   REGION "Manipolatori - Movimento BTrk da Uscita Deposito A0303 alto Vs Uscita deposito A0303 basso"
      "BTrk_Presence"(
         en := TRUE,
         Item := BTrk.A0302_EXIT.B
      );

      "BTrk_Absence"(
         en := "BTrk_Presence"(Item := BTrk.A0302_EXIT.B),
         Item := BTrk.A0302_EXIT.B
      );

      "BTrk_Absence"(
         en := "BTrk_Absence"(Item := BTrk.A0302_EXIT.B),
         Item := BTrk.A0303.Preparation.B
      );

      "BTrk_Presence"(
         en := BTrk.A0302_EXIT.B,
         Item := BTrk.A0302_EXIT.B
      );

      "BTrk_Presence"(Item := BTrk.A0302_EXIT.B);
      IF "BTrk_Presence"(Item := BTrk.A0302_EXIT.B) THEN
         "BTrk_Absence"(Item := BTrk.A0302_EXIT.B);
      END_IF;
      IF "BTrk_Absence"(Item := BTrk.A0302_EXIT.B) THEN
         "BTrk_Absence"(Item := BTrk.A0303.Preparation.B);
      END_IF;
      Ctrl.TRK.BTrk.CheckOut_GoodQlty_UP_To_DOWN := ((("BTrk_Absence"(Item := BTrk.A0303.Preparation.B) AND CIn.Manipolatori.InPos_BancoA0303) AND CIn.Banco_A0303.ReadyToRecive) OR (("BTrk_Absence"(Item := BTrk.A0303.Preparation.B) AND CIn.Manipolatori.InPos_BancoA0303) AND A03_DEBUG.A0302_Manager.A0303_ReadyToRecive));
      IF ((Ctrl.TRK.BTrk.CheckOut_GoodQlty_UP_To_DOWN AND CIn.Manipolatori.Testa.Sollevatore.Work) AND CIn.Manipolatori.Coda.Sollevatore.Work) THEN
         BTrk.A0302_EXIT.B := BTrk.A0302_EXIT.B;
      END_IF;
   END_REGION

   REGION "Manipolatori - Movimento BTrk  Uscita deposito A0303 basso == a ==> Rilascia Beam"
      "BTrk_Presence"(
         en := TRUE,
         Item := BTrk.A0302_EXIT.B
      );

      "BTrk_Absence"(
         en := "BTrk_Presence"(Item := BTrk.A0302_EXIT.B),
         Item := BTrk.A0303.Preparation.B
      );

      "BTrk_Presence"(Item := BTrk.A0302_EXIT.B);
      IF "BTrk_Presence"(Item := BTrk.A0302_EXIT.B) THEN
         "BTrk_Absence"(Item := BTrk.A0303.Preparation.B);
      END_IF;
      Ctrl.TRK.BTrk.CheckOut_GoodQlty_DOWN_To_Sgancia := (((("BTrk_Absence"(Item := BTrk.A0303.Preparation.B) AND CIn.Manipolatori.Testa.Sollevatore.Rest) AND CIn.Manipolatori.Coda.Sollevatore.Rest) AND CIn.Manipolatori.Testa.Sollevatore.Standstill) AND CIn.Manipolatori.Coda.Sollevatore.Standstill);
      IF ((((Ctrl.TRK.BTrk.CheckOut_GoodQlty_DOWN_To_Sgancia AND CIn.Manipolatori.Testa.Magnete.Rest) AND CIn.Manipolatori.Coda.Magnete.Rest) AND NOT (CIn.CarroPareggTesta.Sens.PresenzaMat)) AND NOT (CIn.CarroPareggCoda.Sens.PresenzaMat)) THEN
         BTrk.A0303.Preparation.B := BTrk.A0302_EXIT.B;
      END_IF;
   END_REGION

   REGION "[Ax] Manipolatore - Control - Pos. PRELIEVO su carri pareggiatori"
      "BTrk_Absence"(
         en := TRUE,
         Item := BTrk.A0302_EXIT.B
      );

      "BTrk_Absence"(
         en := "BTrk_Absence"(Item := BTrk.A0302_EXIT.B),
         Item := BTrk.A0302_EXIT.B
      );

      "BTrk_Absence"(
         en := "BTrk_Absence"(Item := BTrk.A0302_EXIT.B),
         Item := BTrk.A0302_EXIT.B
      );

      "BTrk_Absence"(
         en := "BTrk_Absence"(Item := BTrk.A0302_EXIT.B),
         Item := BTrk.A0302_EXIT.B
      );

      "BTrk_Absence"(Item := BTrk.A0302_EXIT.B);
      Ctrl.TRK.BTrk.Manipolatori_Return_ToPrelievo := ((("BTrk_Absence"(Item := BTrk.A0302_EXIT.B) AND NOT (CIn.Manipolatori.InPos_Prelievo)) AND NOT (CIn.CarroPareggCoda.Sens.PresenzaMat)) AND NOT (CIn.CarroPareggTesta.Sens.PresenzaMat));
   END_REGION

   REGION "Manipolatori - Controllo del pezzo sui Magneti - Allarme grave se perdo i sensori presenza"
      "BTrk_Presence"(
         en := TRUE,
         Item := BTrk.A0302_EXIT.B
      );

      "BTrk_Presence"(
         en := TRUE,
         Item := BTrk.A0302_EXIT.B
      );

      "BTrk_Presence"(
         en := TRUE,
         Item := BTrk.A0302_EXIT.B
      );

      #TON_AlarmWrongReadPz_Manip(
         IN := (((((((("BTrk_Presence"(Item := BTrk.A0302_EXIT.B) OR "BTrk_Presence"(Item := BTrk.A0302_EXIT.B) OR "BTrk_Presence"(Item := BTrk.A0302_EXIT.B)) AND CIn.Manipolatori.Testa.Sollevatore.Rest) AND CIn.Manipolatori.Coda.Sollevatore.Rest) AND CIn.Manipolatori.Testa.Magnete.Work) AND CIn.Manipolatori.Coda.Magnete.Work) AND NOT (CIn.CarroPareggCoda.Sens.PresenzaMat)) AND CIn.CarroPareggTesta.Sens.PresenzaMat) OR ((((((("BTrk_Presence"(Item := BTrk.A0302_EXIT.B) OR "BTrk_Presence"(Item := BTrk.A0302_EXIT.B) OR "BTrk_Presence"(Item := BTrk.A0302_EXIT.B)) AND CIn.Manipolatori.Testa.Sollevatore.Rest) AND CIn.Manipolatori.Coda.Sollevatore.Rest) AND CIn.Manipolatori.Testa.Magnete.Work) AND CIn.Manipolatori.Coda.Magnete.Work) AND CIn.CarroPareggCoda.Sens.PresenzaMat) AND NOT (CIn.CarroPareggTesta.Sens.PresenzaMat))),
         PT := T#2S
      );

      "BTrk_Presence"(Item := BTrk.A0302_EXIT.B);
      #TON_AlarmWrongReadPz_Manip.Q;
      IF #TON_AlarmWrongReadPz_Manip.Q THEN
         Alarm.WrongReadPz_ManipBasso := TRUE;
      END_IF;
   END_REGION

   REGION "[Sollevatori] - Manipolatori Testa/Coda - Movimento operazione a lavoro / a riposo"
      "BTrk_Presence"(
         en := TRUE,
         Item := BTrk.A0302_EXIT.B
      );

      "BTrk_Presence"(
         en := TRUE,
         Item := BTrk.A0302_EXIT.B
      );

      "BTrk_Presence"(
         en := TRUE,
         Item := BTrk.A0302_EXIT.B
      );

      "BTrk_Presence"(
         en := CIn.Manipolatori.InPos_BancoA0303,
         Item := BTrk.A0302_EXIT.B
      );

      "BTrk_Presence"(
         en := TRUE,
         Item := BTrk.A0302_EXIT.B
      );

      "BTrk_Presence"(Item := BTrk.A0302_EXIT.B);
      Ctrl.Manipolatori.Sollevatori.Work := ((("BTrk_Presence"(Item := BTrk.A0302_EXIT.B) OR "BTrk_Presence"(Item := BTrk.A0302_EXIT.B) OR "BTrk_Presence"(Item := BTrk.A0302_EXIT.B)) AND CIn.Manipolatori.InPos_Prelievo) OR ("BTrk_Presence"(Item := BTrk.A0302_EXIT.B) AND CIn.Banco_A0303.ReadyToRecive) OR (("BTrk_Presence"(Item := BTrk.A0302_EXIT.B) AND NOT (CIn.Manipolatori.Testa.Magnete.Rest)) AND NOT (CIn.Manipolatori.Coda.Magnete.Rest)));
      IF ((NOT (CIn.Manipolatori.InPos_BancoA0303) AND NOT (CIn.Manipolatori.InPos_Prelievo)) AND NOT (CIn.Manipolatori.InPos_BancoScarto)) THEN
         Ctrl.Manipolatori.Sollevatori.Work := FALSE;
      END_IF;
      Ctrl.Manipolatori.Sollevatori.Rest := NOT (Ctrl.Manipolatori.Sollevatori.Work);
   END_REGION

   REGION "[Magneti] - Manipolatori Testa/Coda - Movimento operazione a lavoro / a riposo"
      "BTrk_Presence"(
         en := TRUE,
         Item := BTrk.A0302_EXIT.B
      );

      "BTrk_Presence"(
         en := TRUE,
         Item := BTrk.A0302_EXIT.B
      );

      "BTrk_Presence"(
         en := TRUE,
         Item := BTrk.A0302_EXIT.B
      );

      "BTrk_Presence"(
         en := TRUE,
         Item := BTrk.A0302_EXIT.B
      );

      "BTrk_Presence"(
         en := TRUE,
         Item := BTrk.A0302_EXIT.B
      );

      "BTrk_Presence"(
         en := TRUE,
         Item := BTrk.A0302_EXIT.B
      );

      "BTrk_Presence"(Item := BTrk.A0302_EXIT.B);
      Ctrl.Manipolatori.Magneti.Work := ((((("BTrk_Presence"(Item := BTrk.A0302_EXIT.B) OR "BTrk_Presence"(Item := BTrk.A0302_EXIT.B)) AND CIn.Manipolatori.InPos_Prelievo) AND CIn.Manipolatori.Testa.Sollevatore.Work) AND CIn.Manipolatori.Coda.Sollevatore.Work) OR "BTrk_Presence"(Item := BTrk.A0302_EXIT.B) OR ("BTrk_Presence"(Item := BTrk.A0302_EXIT.B) AND NOT (CIn.Manipolatori.Testa.Sollevatore.Work)) OR ("BTrk_Presence"(Item := BTrk.A0302_EXIT.B) AND NOT (CIn.Manipolatori.Coda.Sollevatore.Work)) OR ("BTrk_Presence"(Item := BTrk.A0302_EXIT.B) AND NOT (CIn.Manipolatori.InPos_BancoScarto)) OR ("BTrk_Presence"(Item := BTrk.A0302_EXIT.B) AND NOT (CIn.Manipolatori.InPos_BancoA0303)));
      Ctrl.Manipolatori.Magneti.Rest := NOT (Ctrl.Manipolatori.Magneti.Work);
   END_REGION

   REGION "[Sollevatori + Magneti + Ax] - Manipolatori Testa/Coda - COut Manager"
      COut.Manipolatori.Ax.Control_ON := NOT ((NOT (Sts.SemiAut.ON) AND NOT (AreaInterface.Cycle)));
      COut.Manipolatori.Sollevatori.Rest := (NOT ((NOT (Sts.SemiAut.ON) AND NOT (AreaInterface.Cycle))) AND Ctrl.Manipolatori.Sollevatori.Rest);
      COut.Manipolatori.Sollevatori.Work := (NOT ((NOT (Sts.SemiAut.ON) AND NOT (AreaInterface.Cycle))) AND Ctrl.Manipolatori.Sollevatori.Work);
      COut.Manipolatori.Magneti.Rest := (NOT ((NOT (Sts.SemiAut.ON) AND NOT (AreaInterface.Cycle))) AND Ctrl.Manipolatori.Magneti.Rest);
      COut.Manipolatori.Magneti.Work := (NOT ((NOT (Sts.SemiAut.ON) AND NOT (AreaInterface.Cycle))) AND Ctrl.Manipolatori.Magneti.Work);
      COut.Manipolatori.Ax.MoveToPos := ((((COut.Manipolatori.Ax.Control_ON AND Ctrl.TRK.BTrk.CheckOut_BadQlty_UP_MoveToPos) AND NOT (CIn.Manipolatori.InPos_BancoScarto)) OR ((COut.Manipolatori.Ax.Control_ON AND Ctrl.TRK.BTrk.CheckOut_GoodQlty_UP_MoveToPos) AND NOT (CIn.Manipolatori.InPos_BancoA0303)) OR ((COut.Manipolatori.Ax.Control_ON AND Ctrl.TRK.BTrk.Manipolatori_Return_ToPrelievo) AND NOT (CIn.Manipolatori.InPos_Prelievo))) AND NOT (Alarm.WrongReadPz_ManipBasso));
      IF CIn.Manipolatori.InPos_BancoScarto THEN
         Ctrl.TRK.BTrk.PresaAlto_To_CheckOut_BadQlty := FALSE;
      END_IF;
      IF CIn.Manipolatori.InPos_BancoA0303 THEN
         Ctrl.TRK.BTrk.PresaAlto_To_CheckOut_GoodQlty := FALSE;
      END_IF;
      IF CIn.Manipolatori.InPos_Prelievo THEN
         Ctrl.TRK.BTrk.Manipolatori_Return_ToPrelievo := FALSE;
      END_IF;
      COut.Manipolatori.Ax.EnableStopDoorOpeningReq := MachineInterface.MotionsStandStill;
      COut.Manipolatori.Ax.EnableStopInPhase := MachineInterface.AckStopInPhase;
      COut.Manipolatori.Ax.EnableStopProgrammed := MachineInterface.AckStopProgrammed;
   END_REGION

   REGION "[Ax] - Manipolatori Testa/Coda - RIFERIMENTI"
      IF Ctrl.TRK.BTrk.PresaAlto_To_CheckOut_GoodQlty THEN
         COut.Manipolatori.Ax.Pos := A0302_Manipolatore_PERS.Par.Ax_Pos.BancoA0303;
      END_IF;
   END_REGION

   REGION "Stop Cycle"
      #TON_Stop(
         IN := ((AreaInterface.StopProgrammed OR CIn.ProdManager.STOP_FineTurno OR CIn.ProdManager.STOP_ControlloQualita OR AreaInterface.StopInPhase) AND Sts.IsStandstill),
         PT := T#1s
      );

      #TON_Stop.Q;
      Ctrl.Stop := #TON_Stop.Q;
      IF (#TON_Stop.Q AND CIn.ProdManager.STOP_FineTurno) THEN
         Alarm.STOP_FineTurno := TRUE;
      END_IF;
      IF (#TON_Stop.Q AND CIn.ProdManager.STOP_ControlloQualita) THEN
         Alarm.STOP_ControlloQualita := TRUE;
      END_IF;
      IF CIn.ProdManager.STOP_End_Of_Production THEN
         Alarm.STOP_End_Of_Proroduction := TRUE;
      END_IF;
   END_REGION

   REGION "All motions standstill"
      Sts.IsStandstill := ((((((((CIn.P5.SpintoreLong.Ax.Standstill AND CIn.Bordatrice.Ax.Standstill) AND A0302_Bordatrice_RegolazioneFormato.AX_D[1].COut.Standstill) AND CIn.Rulliera.Ax_1.Standstill) AND CIn.Rulliera.Ax_2.Standstill) AND CIn.CarroPareggCoda.Ax.Standstill) AND CIn.CarroPareggTesta.Ax.Standstill) AND CIn.Manipolatori.Testa.Ax.Standstill) AND CIn.Manipolatori.Coda.Ax.Standstill);
   END_REGION

   REGION "Alarms / Warning presence"
      Sts.AlarmsPresence := (NOT ((((NOT (Alarm.WrongReadPz_ManipBasso) AND NOT (Alarm.STOP_End_Of_Proroduction)) AND NOT (Alarm.STOP_ControlloQualita)) AND NOT (Alarm.STOP_FineTurno))) AND NOT (AreaInterface.Man));
      Sts.WarningsPresence := (NOT ((((NOT (Alarm.WrongReadPz_ManipBasso) AND NOT (Alarm.STOP_End_Of_Proroduction)) AND NOT (Alarm.STOP_ControlloQualita)) AND NOT (Alarm.STOP_FineTurno))) AND AreaInterface.Man);
   END_REGION

   REGION "Collect machine to area interface"
      MachineInterface.AlarmsPresence := Sts.AlarmsPresence;

      MachineInterface.WarningPresence := Sts.WarningsPresence;

      MachineInterface.MotionsStandStill := Sts.IsStandstill;

      MachineInterface.AutReady := AreaInterface.Aut AND NOT Sts.AlarmsPresence;


      MachineInterface.AckStopInPhase := AreaInterface.StopInPhase AND Ctrl.Stop;

      MachineInterface.AckStopProgrammed := AreaInterface.StopProgrammed AND Ctrl.Stop;


      MachineInterface.Aborting := AreaInterface.Aut AND Sts.AlarmsPresence;


   END_REGION


END_FUNCTION_BLOCK
